//********************************************************************************
// FUN_PolarToCartesian.
// -------------------------------------------------------------------------------
// This function calculates the cartesian X and Y coordinates from the 
// polar coordinates r and theta.
//	
// Version:
//			- V1.00.00	HHL, 01/04-2021
//********************************************************************************
FUNCTION FUN_PolarToCartesian : BOOL
VAR_IN_OUT
END_VAR
VAR_INPUT
	fRadius			:REAL;			// Radius for polar coordinate
	fAngle			:REAL;			// [deg] Angle for polar coordinate 
END_VAR
VAR_OUTPUT
	fX				:REAL;			// X-axis coordinate
	fY				:REAL;			// Y-axis coordinate	
END_VAR


// Calculate cartesian coordinates from polar coordinates
fX := LREAL_TO_REAL(fRadius * COS(DEG_TO_RAD(fAngle)));
fY := LREAL_TO_REAL(fRadius * SIN(DEG_TO_RAD(fAngle)));

END_FUNCTION

(* stored: Version 1.1.0.1, ProductVersion 3.1.4024.12
   POU FUN_PolarToCartesian: Id {689aba0c-50b6-4c5c-90a1-c84e82e7ff61}, SpecialFunc None *)
